FUNCTION_BLOCK fb_Drehzahl
VAR_INPUT

		TRIGGER : BOOL;	

END_VAR
VAR_OUTPUT
	
	UMDREHUNGEN_PRO_MINUTE : INT;
	
END_VAR
VAR
	
		
	R_TRIG: R_TRIG;
	TON_COUNTER : TON;
	DREHIMPULSE_1S : INT;

END_VAR

R_TRIG(CLK:= TRIGGER);

TON_COUNTER(IN:= NOT TON_COUNTER.Q, PT := T#5S);


IF R_TRIG.Q THEN
	

	DREHIMPULSE_1S := DREHIMPULSE_1S + 1;

END_IF

IF TON_COUNTER.Q THEN
	

	UMDREHUNGEN_PRO_MINUTE := DREHIMPULSE_1S * 12;
	DREHIMPULSE_1S := 0;

END_IF

END_FUNCTION_BLOCK

(* stored: Version 1.1.0.1, ProductVersion 3.1.4024.12
   POU fb_Drehzahl: Id {d26542d3-bdc1-485d-bc40-0654aa42272b}, SpecialFunc None *)
